FUNCTION_BLOCK FB_DeleteFile
VAR_INPUT
	IN_Start				: BOOL;
	IN_Dir					: T_MaxString;
END_VAR
VAR_OUTPUT
	OUT_Error				: BOOL;
	OUT_Busy				: BOOL;
END_VAR
VAR
	
	TrigStart				: R_TRIG;
	RsStart					: RS;
	FileDelete				: FB_FileDelete;
	
	

END_VAR

OUT_Busy := TRUE;

TrigStart(CLK := IN_Start);
FileDelete(sNetId := '', sPathName := IN_Dir, bExecute := TrigStart.Q);

RsStart(SET := TrigStart.Q);
IF RsStart.Q1 THEN
	IF NOT FileDelete.bBusy THEN
		IF FileDelete.bError THEN
			OUT_Error := TRUE;
			OUT_Busy := FALSE;
		ELSE 
			OUT_Error := FALSE;
			OUT_Busy := FALSE;
		END_IF
		TrigStart(CLK := FALSE);
		RsStart(RESET1 := TRUE);
		RsStart(RESET1 := FALSE);
	END_IF
END_IF

END_FUNCTION_BLOCK

(* stored: Version 1.1.0.1, ProductVersion 3.1.4024.6
   POU FB_DeleteFile: Id {9578e081-2a2c-402e-9f5d-e3082ea658e0}, SpecialFunc None *)
